// Mitsubishi GX Works2 project: LRI - PLC - SEM ST V2   PLC: Q03UDV

// task Task_01 (event TRUE, interval 0, priority 31): POU_01

PROGRAM POU_01
VAR
  i_EstadoSemafaro : ARRAY [0..9] OF INT;
  stSemafaro_1 : stSemafaro;
END_VAR
stSemafaro_1();
END_PROGRAM

FUNCTION_BLOCK stSemafaro
VAR_OUTPUT
  o_Verde1 : BOOL;
  o_Amarelo1 : BOOL;
  o_Vermelho1 : BOOL;
  o_Verde2 : BOOL;
  o_Amarelo2 : BOOL;
  o_Vermelho2 : BOOL;
END_VAR
VAR
  x_timer : INT;
  i_Auxiliar : ARRAY [0..599] OF INT;
END_VAR
IF x_timer <= 551THEN
	FOR x_timer := 0 TO 551 BY 1 DO
		i_Auxiliar[x_timer]:= x_timer+1;

		CASE x_timer OF
			0, 100:
			o_Verde1 		:= 1;
			o_Amarelo1 	:= 0;
			o_Vermelho1 := 0;
			o_Verde2		 	:= 0;
			o_Amarelo2 	:= 0;
			o_Vermelho2 := 1;
			
			101, 110:
			o_Verde1	:= 0;
			
			111, 120:
			o_Verde1	:= 1;
			
			121, 130:
			o_Verde1	:= 0;
			
			131, 140:
			o_Verde1	:= 1;
			
			141, 150:
			o_Verde1	:= 0;
			
			161, 170:
			o_Verde1	:= 1;
			
			171, 180:
			o_Verde1	:= 0;
			
			181, 190:
			o_Verde1	:= 1;
			
			191, 200:
			o_Verde1	:= 0;
			
			201, 300:
			o_Verde1 		:= 0;
			o_Amarelo1 	:= 1;
			o_Vermelho1 := 0;
			o_Verde2		 	:= 0;
			o_Amarelo2 	:= 0;
			o_Vermelho2 := 1;
			
			301, 350:
			o_Verde1 		:= 0;
			o_Amarelo1 	:= 0;
			o_Vermelho1 := 1;
			o_Verde2		 	:= 0;
			o_Amarelo2 	:= 0;
			o_Vermelho2 := 1;
			
			351, 450:
			o_Verde1 		:= 0;
			o_Amarelo1 	:= 0;
			o_Vermelho1 := 1;
			o_Verde2		 	:= 1;
			o_Amarelo2 	:= 0;
			o_Vermelho2 := 0;
			
			451, 460:
			o_Verde2	:= 0;
			
			461, 470:
			o_Verde2	:= 1;
			
			471, 480:
			o_Verde2	:= 0;
			
			481, 490:
			o_Verde2	:= 1;
			
			501, 510:
			o_Verde2	:= 0;
			
			511,520:
			o_Verde2	:= 1;
			
			521, 530:
			o_Verde2	:= 0;
			
			531, 540:
			o_Verde2	:= 1;
			
			541, 550:
			o_Verde2	:= 0;
			
			351, 450:
			o_Verde1 		:= 0;
			o_Amarelo1 	:= 0;
			o_Vermelho1 := 1;
			o_Verde2		 	:= 0;
			o_Amarelo2 	:= 1;
			o_Vermelho2 := 0;
			
			451, 550:
			o_Verde1 		:= 0;
			o_Amarelo1 	:= 0;
			o_Vermelho1 := 1;
			o_Verde2		 	:= 0;
			o_Amarelo2 	:= 0;
			o_Vermelho2 := 1;
			
		END_CASE;	
			IF x_timer >= 550THEN
					i_Auxiliar[x_timer]:= 0;
			END_IF;
		
	END_FOR;
END_IF;
END_FUNCTION_BLOCK
